// TIA Portal V17 export
// export: Created 2025-06-25T13:13:25.9235506Z, ExportSetting WithDefaults, DisplayName Totally Integrated Automation Portal, DisplayVersion V17 Update 8, DisplayName TIA Portal Openness, DisplayVersion V17 Update 8, DisplayName TIA Portal Version Control Interface, DisplayVersion V17, DisplayName STEP 7 Professional, DisplayVersion V17 Update 8, DisplayName STEP 7 Safety, DisplayVersion V17 Update 6, DisplayName WinCC Advanced, DisplayVersion V17 Update 8
DATA_BLOCK "DB_AI"   // DB40
{ S7_Optimized_Access := 'FALSE' }
AUTHOR : Heaten
VERSION : 0.1
// stored: AutoNumber true, DBAccessibleFromOPCUA true, DBAccessibleFromWebserver true, IsOnlyStoredInLoadMemory false, IsWriteProtectedInAS false
   VAR RETAIN
      HBL_TT_502 { S7_SetPoint := 'True'} : "stAnalogInput";   // Compressor discharge popoff temperature
      HBL_PT_503 { S7_SetPoint := 'True'} : "stAnalogInput";   // Compressor discharge pressure
      HBL_TT_504 { S7_SetPoint := 'True'} : "stAnalogInput";   // Compressor discharge temperature
      HBL_TT_505 { S7_SetPoint := 'True'} : "stAnalogInput";   // Compressor discharge temperature
      HBL_PT_506 { S7_SetPoint := 'True'} : "stAnalogInput";   // Compressor discharge pressure
      HBL_LT_510 { S7_SetPoint := 'True'} : "stAnalogInput";   // Steam generator condensate level
      HBL_PT_511 { S7_SetPoint := 'True'} : "stAnalogInput";   // Heat sink discharge pressure
      HBL_TT_512 { S7_SetPoint := 'True'} : "stAnalogInput";   // Heat sink discharge temperature
      HBL_TT_516 { S7_SetPoint := 'True'} : "stAnalogInput";   // Steam generator suction temperature
      HBL_PT_517 { S7_SetPoint := 'True'} : "stAnalogInput";   // Steam generator suction pressure
      HBL_TT_518 { S7_SetPoint := 'True'} : "stAnalogInput";   // Heat sink discharge process temperature
      HBL_PT_519 { S7_SetPoint := 'True'} : "stAnalogInput";   // Heat sink discharge process pressure
      HBL_FT_520 { S7_SetPoint := 'True'} : "stAnalogInput";   // Refrigerant flow
      HBL_CT_524 { S7_SetPoint := 'True'} : "stAnalogInput";   // Gas detector steam generator suction popoff
      HBL_TT_525 { S7_SetPoint := 'True'} : "stAnalogInput";   // Steam generator (condenser) suction temperature
      HBL_PT_526 { S7_SetPoint := 'True'} : "stAnalogInput";   // Steam generator (condenser) suction pressure
      HBL_FT_527 { S7_SetPoint := 'True'} : "stAnalogInput";   // Heat sink condensate blowdown flow
      HBL_TT_530 { S7_SetPoint := 'True'} : "stAnalogInput";   // Expansion valve B discharge temperature
      HBL_PT_531 { S7_SetPoint := 'True'} : "stAnalogInput";   // Expansion valve B discharge pressure
      HBL_TT_532 { S7_SetPoint := 'True'} : "stAnalogInput";   // Heat source 1 discharge temperature
      HBL_TT_533 { S7_SetPoint := 'True'} : "stAnalogInput";   // Evaporator 1 discharge temperature
      HBL_PT_534 { S7_SetPoint := 'True'} : "stAnalogInput";   // Evaporator 1 discharge pressure
      HBL_AT_535 { S7_SetPoint := 'True'} : "stAnalogInput";   // Evaporator 1 steam quality
      HBL_CT_538 { S7_SetPoint := 'True'} : "stAnalogInput";   // Gas detector evaporator popoff
      HBL_TT_540 { S7_SetPoint := 'True'} : "stAnalogInput";   // Expansion valve A discharge temperature
      HBL_PT_541 { S7_SetPoint := 'True'} : "stAnalogInput";   // Expansion valve A discharge pressure
      HBL_TT_542 { S7_SetPoint := 'True'} : "stAnalogInput";   // Heat source 2 discharge temperature
      HBL_TT_543 { S7_SetPoint := 'True'} : "stAnalogInput";   // Evaporator 2 discharge temperature
      HBL_PT_544 { S7_SetPoint := 'True'} : "stAnalogInput";   // Evaporator 2 discharge pressure
      HBL_AT_545 { S7_SetPoint := 'True'} : "stAnalogInput";   // Evaporator 2 steam quality
      HBL_TT_546 { S7_SetPoint := 'True'} : "stAnalogInput";   // Heat source suction temperature
      HBL_PT_547 { S7_SetPoint := 'True'} : "stAnalogInput";   // Heast source suction pressure
      HBL_PT_561 { S7_SetPoint := 'True'} : "stAnalogInput";   // Evaporator 1 axis A vacuum pressure
      HBL_PT_562 { S7_SetPoint := 'True'} : "stAnalogInput";   // Evaporator 2 axis A vacuum pressure
      HBL_FT_565 { S7_SetPoint := 'True'} : "stAnalogInput";   // Heat source 1 discharge condensate flow
      HBL_FT_566 { S7_SetPoint := 'True'} : "stAnalogInput";   // Heat source 2 discharge condensate flow
      HBL_TT_571 { S7_SetPoint := 'True'} : "stAnalogInput";   // Compressor suction temperature
      HBL_PT_572 { S7_SetPoint := 'True'} : "stAnalogInput";   // Compressor suction pressure
      HBL_TT_573 { S7_SetPoint := 'True'} : "stAnalogInput";   // Expansion valve suction temperature
      HBL_PT_580 { S7_SetPoint := 'True'} : "stAnalogInput";   // Expansion valve suction pressure
      HBL_LT_610 { S7_SetPoint := 'True'} : "stAnalogInput";   // HP receiver refrigerant level
      HBL_TT_611 { S7_SetPoint := 'True'} : "stAnalogInput";   // Steam generator discharge temperature
      HBL_PT_612 { S7_SetPoint := 'True'} : "stAnalogInput";   // Steam generator discharge pressure
      HBL_CT_615 { S7_SetPoint := 'True'} : "stAnalogInput";   // Gas detector PSV discharge pipe
      HBL_PT_618 { S7_SetPoint := 'True'} : "stAnalogInput";   // HP Receiver pressure
      HBL_CT_620 { S7_SetPoint := 'True'} : "stAnalogInput";   // Gas detector recuperator popoff
      HBL_PT_635 { S7_SetPoint := 'True'} : "stAnalogInput";   // Oil separator stage 1 oil return pressure
      HBL_PT_636 { S7_SetPoint := 'True'} : "stAnalogInput";   // Oil separator stage 2 oil return pressure
      HBL_CT_643 { S7_SetPoint := 'True'} : "stAnalogInput";   // Gas detector suction accumulator popoff
      HBL_LT_650 { S7_SetPoint := 'True'} : "stAnalogInput";   // Heat source condensate buffer tank level
      HBL_CT_673 { S7_SetPoint := 'True'} : "stAnalogInput";   // Gas detector oil separator discharge popoff
      HBL_PT_651 { S7_SetPoint := 'True'} : "stAnalogInput";   // Heat source condensate buffer tank pressure
      HBL_PT_701 { S7_SetPoint := 'True'} : "stAnalogInput";   // Filter dryer suction pressure
      HBL_PT_702 { S7_SetPoint := 'True'} : "stAnalogInput";   // Filter dryer discharge pressure
      HBL_PT_703 { S7_SetPoint := 'True'} : "stAnalogInput";   // Filter dryer differential pressure
      CPC_CT_851 { S7_SetPoint := 'True'} : "stAnalogInput";   // Gas detector CPC popoff
      CPC_PT_862 { S7_SetPoint := 'True'} : "stAnalogInput";   // CPC pump discharge pressure
      CPC_PT_865 { S7_SetPoint := 'True'} : "stAnalogInput";   // CPC pump suction pressure
      CPC_TT_866 { S7_SetPoint := 'True'} : "stAnalogInput";   // CPC pump suction temperature
      CPC_LT_870 { S7_SetPoint := 'True'} : "stAnalogInput";   // CPC tank refrigerant level
      CPC_TT_871 { S7_SetPoint := 'True'} : "stAnalogInput";   // CPC tank refrigerant temperature
      CPC_PT_872 { S7_SetPoint := 'True'} : "stAnalogInput";   // CPC tank refrigerant pressure
      HBL_TT_901 { S7_SetPoint := 'True'} : "stAnalogInput";   // Heat sink suction temperature
      HBL_PT_902 { S7_SetPoint := 'True'} : "stAnalogInput";   // Heat sink suction pressure
      HBL_TT_03 { S7_SetPoint := 'True'} : "stAnalogInput";   // Oil sump oil temperature
      HBL_TT_16 { S7_SetPoint := 'True'} : "stAnalogInput";   // Container air temperature
      HBL_TT_17 { S7_SetPoint := 'True'} : "stAnalogInput";   // Control cabinet air temperature
      HBL_TT_18 { S7_SetPoint := 'True'} : "stAnalogInput";   // Ambient air temperature
      HBL_TT_20 { S7_SetPoint := 'True'} : "stAnalogInput";   // Compressor motor winding temperature
      HBL_TT_21 { S7_SetPoint := 'True'} : "stAnalogInput";   // Oil sump wall temperature left
      HBL_TT_22 { S7_SetPoint := 'True'} : "stAnalogInput";   // Oil sump wall temperature right
      HBL_TT_23 { S7_SetPoint := 'True'} : "stAnalogInput";   // Compressor motor U-winding temperature
      HBL_TT_24 { S7_SetPoint := 'True'} : "stAnalogInput";   // Compressor motor V-winding temperature
      HBL_TT_25 { S7_SetPoint := 'True'} : "stAnalogInput";   // Compressor motor W-winding temperature
      HBL_TT_26 { S7_SetPoint := 'True'} : "stAnalogInput";   // Compressor motor D bearing temperature
      HBL_TT_27 { S7_SetPoint := 'True'} : "stAnalogInput";   // Compressor motor N bearing temperature
      HBL_PT_05 { S7_SetPoint := 'True'} : "stAnalogInput";   // Crankcase gas pressure
      HBL_PT_960 { S7_SetPoint := 'True'} : "stAnalogInput";   // Oil pump discharge pressure
      HBL_PT_961 { S7_SetPoint := 'True'} : "stAnalogInput";   // Oil gallery pressure
      HBL_CT_01 { S7_SetPoint := 'True'} : "stAnalogInput";   // Gas detector Heatbooster (optional)
      HBL_CT_950 { S7_SetPoint := 'True'} : "stAnalogInput";   // Gas detector container/compressor room
      SSC_TT_01 { S7_SetPoint := 'True'} : "stAnalogInput";   // SSC seal suction temperature
      SSC_TT_02 { S7_SetPoint := 'True'} : "stAnalogInput";   // SSC seal discharge temperature
      SSC_TT_03 { S7_SetPoint := 'True'} : "stAnalogInput";   // SSC barrier fluid circulation pump suction temperature
      SSC_TT_04 { S7_SetPoint := 'True'} : "stAnalogInput";   // SSC barrier fluid heat exchanger temperature
      SSC_PIT_01 { S7_SetPoint := 'True'} : "stAnalogInput";   // SSC barrier fluid accumulator pressure
      SSC_PDT_01 { S7_SetPoint := 'True'} : "stAnalogInput";   // SSC barrier fluid circulation pump differential pressure
      SSC_LT_01 { S7_SetPoint := 'True'} : "stAnalogInput";   // SSC barrier fluid reservoir level
      Spare { S7_SetPoint := 'True'} : "stAnalogInput";
   END_VAR
BEGIN
   HBL_TT_502.Raw.iMin := -14500;
   HBL_TT_502.Raw.iMax := 15500;
   HBL_TT_502.Eng.fMin := -145.0;
   HBL_TT_502.Eng.fMax := 155.0;
   HBL_PT_503.Raw.iMin := 0;
   HBL_PT_503.Raw.iMax := 27648;
   HBL_PT_503.Eng.fMin := 0.0;
   HBL_PT_503.Eng.fMax := 6000.0;
   HBL_TT_504.Raw.iMin := -14500;
   HBL_TT_504.Raw.iMax := 15500;
   HBL_TT_504.Eng.fMin := -145.0;
   HBL_TT_504.Eng.fMax := 155.0;
   HBL_TT_505.Raw.iMin := -14500;
   HBL_TT_505.Raw.iMax := 15500;
   HBL_TT_505.Eng.fMin := -145.0;
   HBL_TT_505.Eng.fMax := 155.0;
   HBL_PT_506.Eng.fMin := 0.0;
   HBL_PT_506.Eng.fMax := 2500.0;
   HBL_LT_510.Raw.iMin := 0;
   HBL_LT_510.Raw.iMax := 27648;
   HBL_LT_510.Eng.fMin := 0.0;
   HBL_LT_510.Eng.fMax := 100.0;
   HBL_PT_511.Raw.iMin := 0;
   HBL_PT_511.Raw.iMax := 27648;
   HBL_PT_511.Eng.fMin := 0.0;
   HBL_PT_511.Eng.fMax := 4000.0;
   HBL_TT_512.Raw.iMin := -14500;
   HBL_TT_512.Raw.iMax := 15500;
   HBL_TT_512.Eng.fMin := -145.0;
   HBL_TT_512.Eng.fMax := 155.0;
   HBL_TT_516.Raw.iMin := -14500;
   HBL_TT_516.Raw.iMax := 15500;
   HBL_TT_516.Eng.fMin := -145.0;
   HBL_TT_516.Eng.fMax := 155.0;
   HBL_PT_517.Raw.iMin := 0;
   HBL_PT_517.Raw.iMax := 27648;
   HBL_PT_517.Eng.fMax := 4000.0;
   HBL_TT_518.Raw.iMin := -14500;
   HBL_TT_518.Raw.iMax := 15500;
   HBL_TT_518.Eng.fMin := -145.0;
   HBL_TT_518.Eng.fMax := 155.0;
   HBL_PT_519.Raw.iMax := 27648;
   HBL_PT_519.Eng.fMax := 2500.0;
   HBL_FT_520.Raw.iMin := 0;
   HBL_FT_520.Raw.iMax := 27648;
   HBL_FT_520.Eng.fMin := 0.0;
   HBL_FT_520.Eng.fMax := 16.667;
   // HBL_FT_520.Eng.fValue : [L/s]
   HBL_CT_524.Eng.fMin := 0.0;
   HBL_CT_524.Eng.fMax := 5000.0;
   HBL_TT_525.Raw.iMin := -14500;
   HBL_TT_525.Raw.iMax := 15500;
   HBL_TT_525.Eng.fMin := -145.0;
   HBL_TT_525.Eng.fMax := 155.0;
   HBL_PT_526.Raw.iMax := 27648;
   HBL_PT_526.Eng.fMax := 4000.0;
   HBL_TT_530.Raw.iMin := -14500;
   HBL_TT_530.Raw.iMax := 15500;
   HBL_TT_530.Eng.fMin := -145.0;
   HBL_TT_530.Eng.fMax := 155.0;
   HBL_PT_531.Raw.iMin := 0;
   HBL_PT_531.Raw.iMax := 27648;
   HBL_PT_531.Eng.fMin := 0.0;   // [kPa]
   HBL_PT_531.Eng.fMax := 3450.0;   // [kPa]
   HBL_TT_532.Raw.iMin := -14500;
   HBL_TT_532.Raw.iMax := 15500;
   HBL_TT_532.Eng.fMin := -145.0;
   HBL_TT_532.Eng.fMax := 155.0;
   HBL_TT_533.Raw.iMin := -14500;
   HBL_TT_533.Raw.iMax := 15500;
   HBL_TT_533.Eng.fMin := -145.0;
   HBL_TT_533.Eng.fMax := 155.0;
   HBL_PT_534.Raw.iMin := 0;
   HBL_PT_534.Raw.iMax := 27648;
   HBL_PT_534.Eng.fMin := 0.0;   // [kPa]
   HBL_PT_534.Eng.fMax := 3450.0;   // [kPa]
   HBL_AT_535.Raw.iMin := 0;
   HBL_AT_535.Raw.iMax := 27648;
   HBL_AT_535.Eng.fMin := 0.84;
   HBL_AT_535.Eng.fMax := 1.05;
   HBL_CT_538.Eng.fMin := 0.0;
   HBL_CT_538.Eng.fMax := 5000.0;
   HBL_TT_540.Raw.iMin := -14500;
   HBL_TT_540.Raw.iMax := 15500;
   HBL_TT_540.Eng.fMin := -145.0;
   HBL_TT_540.Eng.fMax := 155.0;
   HBL_PT_541.Raw.iMin := 0;
   HBL_PT_541.Raw.iMax := 27648;
   HBL_PT_541.Eng.fMin := 0.0;   // [kPa]
   HBL_PT_541.Eng.fMax := 3450.0;   // [kPa]
   HBL_TT_542.Raw.iMin := -14500;
   HBL_TT_542.Raw.iMax := 15500;
   HBL_TT_542.Eng.fMin := -145.0;
   HBL_TT_542.Eng.fMax := 155.0;
   HBL_TT_543.Raw.iMin := -14500;
   HBL_TT_543.Raw.iMax := 15500;
   HBL_TT_543.Eng.fMin := -145.0;
   HBL_TT_543.Eng.fMax := 155.0;
   HBL_PT_544.Raw.iMax := 27648;
   HBL_PT_544.Eng.fMin := 0.0;   // [kPa]
   HBL_PT_544.Eng.fMax := 3450.0;   // [kPa]
   HBL_AT_545.Raw.iMin := 0;
   HBL_AT_545.Raw.iMax := 27648;
   HBL_AT_545.Eng.fMin := 0.84;
   HBL_AT_545.Eng.fMax := 1.05;
   HBL_TT_546.Raw.iMin := -14500;
   HBL_TT_546.Raw.iMax := 15500;
   HBL_TT_546.Eng.fMin := -145.0;
   HBL_TT_546.Eng.fMax := 155.0;
   HBL_PT_547.Raw.iMin := 0;
   HBL_PT_547.Raw.iMax := 27648;
   HBL_PT_547.Eng.fMin := 0.0;
   HBL_PT_547.Eng.fMax := 2500.0;
   HBL_PT_561.Eng.fMin := 0.0;
   HBL_PT_561.Eng.fMax := 200.0;
   HBL_PT_562.Eng.fMin := 0.0;
   HBL_PT_562.Eng.fMax := 200.0;
   HBL_FT_565.Eng.fMin := 0.0;
   HBL_FT_565.Eng.fMax := 100.0;
   HBL_FT_566.Eng.fMin := 0.0;
   HBL_FT_566.Eng.fMax := 100.0;
   HBL_TT_571.Raw.iMin := -14500;
   HBL_TT_571.Raw.iMax := 15500;
   HBL_TT_571.Eng.fMin := -145.0;
   HBL_TT_571.Eng.fMax := 155.0;
   HBL_PT_572.Raw.iMin := 0;
   HBL_PT_572.Raw.iMax := 27648;
   HBL_PT_572.Eng.fMin := 0.0;
   HBL_PT_572.Eng.fMax := 4000.0;
   HBL_TT_573.Raw.iMin := -14500;
   HBL_TT_573.Raw.iMax := 15500;
   HBL_TT_573.Eng.fMin := -145.0;
   HBL_TT_573.Eng.fMax := 155.0;
   HBL_PT_580.Eng.fMin := 0.0;
   HBL_PT_580.Eng.fMax := 4000.0;
   HBL_LT_610.Raw.iMin := 0;
   HBL_LT_610.Raw.iMax := 27648;
   HBL_LT_610.Eng.fMin := 0.0;
   HBL_LT_610.Eng.fMax := 100.0;
   HBL_TT_611.Raw.iMin := -14500;
   HBL_TT_611.Raw.iMax := 15500;
   HBL_TT_611.Eng.fMin := -145.0;
   HBL_TT_611.Eng.fMax := 155.0;
   HBL_PT_612.Raw.iMax := 27648;
   HBL_PT_612.Eng.fMax := 4000.0;
   HBL_CT_615.Raw.iMin := 0;
   HBL_CT_615.Raw.iMax := 27648;
   HBL_CT_615.Eng.fMin := 0.0;
   HBL_CT_615.Eng.fMax := 2000.0;
   HBL_PT_618.Raw.iMin := 0;
   HBL_PT_618.Raw.iMax := 27648;
   HBL_PT_618.Eng.fMin := 0.0;
   HBL_PT_618.Eng.fMax := 3450.0;
   HBL_CT_620.Eng.fMin := 0.0;
   HBL_CT_620.Eng.fMax := 5000.0;
   HBL_PT_635.Raw.iMin := 0;
   HBL_PT_635.Raw.iMax := 27648;
   HBL_PT_635.Eng.fMin := 0.0;   // [kPa]
   HBL_PT_635.Eng.fMax := 3450.0;   // [kPa]
   HBL_PT_636.Raw.iMin := 0;
   HBL_PT_636.Raw.iMax := 27648;
   HBL_PT_636.Eng.fMin := 0.0;   // [kPa]
   HBL_PT_636.Eng.fMax := 3450.0;   // [kPa]
   HBL_CT_643.Eng.fMin := 0.0;
   HBL_CT_643.Eng.fMax := 5000.0;
   HBL_LT_650.Raw.iMin := 0;
   HBL_LT_650.Raw.iMax := 27648;
   HBL_LT_650.Eng.fMin := 0.0;
   HBL_LT_650.Eng.fMax := 100.0;
   HBL_CT_673.Eng.fMin := 0.0;
   HBL_CT_673.Eng.fMax := 5000.0;
   HBL_PT_651.Raw.iMin := 0;
   HBL_PT_651.Raw.iMax := 27648;
   HBL_PT_651.Eng.fMin := -10.0;   // [kPa]
   HBL_PT_651.Eng.fMax := 1000.0;   // [kPa]
   HBL_PT_701.Raw.iMin := 0;
   HBL_PT_701.Raw.iMax := 27648;
   HBL_PT_701.Eng.fMin := 0.0;
   HBL_PT_701.Eng.fMax := 3450.0;
   HBL_PT_702.Raw.iMin := 0;
   HBL_PT_702.Raw.iMax := 27648;
   HBL_PT_702.Eng.fMin := 0.0;
   HBL_PT_702.Eng.fMax := 3450.0;
   CPC_CT_851.Eng.fMin := 0.0;
   CPC_CT_851.Eng.fMax := 5000.0;
   CPC_PT_862.Raw.iMax := 27648;
   CPC_PT_862.Eng.fMin := 0.0;
   CPC_PT_862.Eng.fMax := 6000.0;
   CPC_PT_865.Eng.fMin := 0.0;
   CPC_PT_865.Eng.fMax := 1600.0;
   CPC_TT_866.Raw.iMin := -14500;
   CPC_TT_866.Raw.iMax := 15500;
   CPC_TT_866.Eng.fMin := -145.0;
   CPC_TT_866.Eng.fMax := 155.0;
   CPC_LT_870.Raw.iMax := 27648;
   CPC_LT_870.Eng.fMax := 100.0;
   CPC_TT_871.Raw.iMin := -14500;
   CPC_TT_871.Raw.iMax := 15500;
   CPC_TT_871.Eng.fMin := -145.0;
   CPC_TT_871.Eng.fMax := 155.0;
   CPC_PT_872.Raw.iMin := 0;
   CPC_PT_872.Raw.iMax := 27648;
   CPC_PT_872.Eng.fMin := 0.0;
   CPC_PT_872.Eng.fMax := 3450.0;
   HBL_TT_901.Raw.iMin := -14500;
   HBL_TT_901.Raw.iMax := 15500;
   HBL_TT_901.Eng.fMin := -145.0;
   HBL_TT_901.Eng.fMax := 155.0;
   HBL_PT_902.Raw.iMin := 0;
   HBL_PT_902.Raw.iMax := 27648;
   HBL_PT_902.Eng.fMin := 0.0;
   HBL_PT_902.Eng.fMax := 2500.0;
   HBL_TT_03.Raw.iMin := -14500;
   HBL_TT_03.Raw.iMax := 15500;
   HBL_TT_03.Eng.fMin := -145.0;
   HBL_TT_03.Eng.fMax := 155.0;
   HBL_TT_16.Raw.iMin := -14500;
   HBL_TT_16.Raw.iMax := 15500;
   HBL_TT_16.Eng.fMin := -145.0;
   HBL_TT_16.Eng.fMax := 155.0;
   HBL_TT_17.Raw.iMin := -14500;
   HBL_TT_17.Raw.iMax := 15500;
   HBL_TT_17.Eng.fMin := -145.0;
   HBL_TT_17.Eng.fMax := 155.0;
   HBL_TT_18.Raw.iMin := -14500;
   HBL_TT_18.Raw.iMax := 15500;
   HBL_TT_18.Eng.fMin := -145.0;
   HBL_TT_18.Eng.fMax := 155.0;
   HBL_TT_20.Raw.iMin := -14500;
   HBL_TT_20.Raw.iMax := 15500;
   HBL_TT_20.Eng.fMin := -145.0;
   HBL_TT_20.Eng.fMax := 155.0;
   HBL_TT_21.Raw.iMin := -14500;
   HBL_TT_21.Raw.iMax := 15500;
   HBL_TT_21.Eng.fMin := -145.0;
   HBL_TT_21.Eng.fMax := 155.0;
   HBL_TT_22.Raw.iMin := -14500;
   HBL_TT_22.Raw.iMax := 15500;
   HBL_TT_22.Eng.fMin := -145.0;
   HBL_TT_22.Eng.fMax := 155.0;
   HBL_TT_23.Raw.iMin := -14500;
   HBL_TT_23.Raw.iMax := 15500;
   HBL_TT_23.Eng.fMin := -145.0;
   HBL_TT_23.Eng.fMax := 155.0;
   HBL_TT_24.Raw.iMin := -14500;
   HBL_TT_24.Raw.iMax := 15500;
   HBL_TT_24.Eng.fMin := -145.0;
   HBL_TT_24.Eng.fMax := 155.0;
   HBL_TT_25.Raw.iMin := -14500;
   HBL_TT_25.Raw.iMax := 15500;
   HBL_TT_25.Eng.fMin := -145.0;
   HBL_TT_25.Eng.fMax := 155.0;
   HBL_TT_26.Raw.iMin := -14500;
   HBL_TT_26.Raw.iMax := 15500;
   HBL_TT_26.Eng.fMin := -145.0;
   HBL_TT_26.Eng.fMax := 155.0;
   HBL_TT_27.Raw.iMin := -14500;
   HBL_TT_27.Raw.iMax := 15500;
   HBL_TT_27.Eng.fMin := -145.0;
   HBL_TT_27.Eng.fMax := 155.0;
   HBL_PT_05.Raw.iMax := 27648;
   HBL_PT_05.Eng.fMax := 2500.0;
   HBL_PT_960.Raw.iMax := 27648;
   HBL_PT_960.Eng.fMax := 2500.0;
   HBL_PT_961.Raw.iMin := 0;
   HBL_PT_961.Raw.iMax := 27648;
   HBL_PT_961.Eng.fMin := 0.0;
   HBL_PT_961.Eng.fMax := 2500.0;
   HBL_CT_01.Raw.iMin := 0;
   HBL_CT_01.Raw.iMax := 27648;
   HBL_CT_01.Eng.fMin := 0.0;
   HBL_CT_01.Eng.fMax := 5000.0;
   HBL_CT_950.Raw.iMin := 0;
   HBL_CT_950.Raw.iMax := 27648;
   HBL_CT_950.Eng.fMin := 0.0;
   HBL_CT_950.Eng.fMax := 2000.0;
   SSC_TT_01.Raw.iMin := -14500;
   SSC_TT_01.Raw.iMax := 15500;
   SSC_TT_01.Eng.fMin := -145.0;
   SSC_TT_01.Eng.fMax := 155.0;
   SSC_TT_02.Raw.iMin := -14500;
   SSC_TT_02.Raw.iMax := 15500;
   SSC_TT_02.Eng.fMin := -145.0;
   SSC_TT_02.Eng.fMax := 155.0;
   SSC_TT_03.Raw.iMin := -14500;
   SSC_TT_03.Raw.iMax := 15500;
   SSC_TT_03.Eng.fMin := -145.0;
   SSC_TT_03.Eng.fMax := 155.0;
   SSC_TT_04.Raw.iMin := -14500;
   SSC_TT_04.Raw.iMax := 15500;
   SSC_TT_04.Eng.fMin := -145.0;
   SSC_TT_04.Eng.fMax := 155.0;
   SSC_PIT_01.Raw.iMin := 0;
   SSC_PIT_01.Raw.iMax := 27648;
   SSC_PIT_01.Eng.fMin := 0.0;
   SSC_PIT_01.Eng.fMax := 2500.0;
   SSC_PDT_01.Raw.iMin := 0;
   SSC_PDT_01.Raw.iMax := 27648;
   SSC_PDT_01.Eng.fMin := 0.0;
   SSC_PDT_01.Eng.fMax := 250.0;
   SSC_LT_01.Raw.iMin := 0;
   SSC_LT_01.Raw.iMax := 27648;
   SSC_LT_01.Eng.fMin := 0.0;
   SSC_LT_01.Eng.fMax := 100.0;
END_DATA_BLOCK
